// Mitsubishi GX Works2 project: PLC_V3   PLC: FX3G

TYPE ST_STEP : STRUCT
  iEnable : INT;  (* Шаг включён (1 - активен) *)
  iRiseTime : INT;  (* Время подъёма, мин *)
  iHoldTime : INT;  (* Время выдержки, мин *)
  iHoldTempr : INT;  (* Уставка температуры выдержки *)
  iHoldHumid : INT;  (* Уставка влажности выдержки *)
  iVFDSpeed : INT;  (* Скорость ПЧ, % *)
END_STRUCT END_TYPE

TYPE ST_STEPHelper : STRUCT
  iState : INT;  (* Состояние шага: 0 - ожидание, 1 - подъём, 2 - выдержка, 3 - завершено *)
END_STRUCT END_TYPE

TYPE ST_VFD : STRUCT
  xEnable : BOOL;  (* Активация ПЧ (разрешение работы) *)
  xManStart : BOOL;  (* Пуск в ручном режиме *)
  iManSpeed : INT;  (* Скорость в ручном режиме (0-500 = 0.0-50.0 Гц) *)
  iState : INT;  (* Текущее состояние ПЧ (0-3) *)
END_STRUCT END_TYPE

// global labels: GVL
VAR_GLOBAL
  grSteps : ARRAY [0..4] OF ST_STEP;  (* Массив шагов программы сушки (5 шагов) / Назначить R1 как главный *)
  griTLimit AT R31 : INT;  (* Дельта ограничения для ПИД температуры *)
  griHLimit AT R32 : INT;  (* Дельта ограничения для ПИД влажности *)
  griMinVentSpeed AT R33 : INT;  (* Минимальная скорость вентилятора влажности, % *)
  griMinVentDelay AT R34 : INT;  (* Мин. задержка перед включением вентилятора после обнуления ПИД, мин *)
  garstStepHelper : ARRAY [0..4] OF ST_STEPHelper;  (* Массив состояния шагов программы (5 шагов) / Назначить D1090 как главный *)
  grVFD : ARRAY [0..14] OF ST_VFD;  (* Массив ПЧ: [0..13] = ПЧ1-14, [14] = ПЧ ВЕНТ / Назначить M420 D1060 как главный *)
  gxReset AT M400 : BOOL;  (* Сброс *)
  gxStart AT M401 : BOOL;  (* Пуск *)
  gxPIDANTemp AT M402 : BOOL;  (* Включить автонастройку ПИД температуры *)
  gxPIDANHum AT M403 : BOOL;  (* Включить автонастройку ПИД влажности *)
  gxPIDANModeTemp AT M404 : BOOL;  (* 0 - предельный цикл, 1 - ступенчатый отклик *)
  gxPIDANModeHum AT M405 : BOOL;  (* 0 - предельный цикл, 1 - ступенчатый отклик *)
  gxDone AT M406 : BOOL;  (* Процесс сушки завершён *)
  gxAlarmReset AT M407 : BOOL;  (* Сброс аварий *)
  gxProgress AT M408 : BOOL;  (* Процесс сушки выполняется *)
  gxPause AT M409 : BOOL;  (* Процесс сушки на паузе (шаг 40) *)
  gxValve1Work AT M410 : BOOL;  (* Клапан 1 в работе (AO_Valve1 > 0) *)
  gxValve2Work AT M411 : BOOL;  (* Клапан 2 в работе (AO_Valve2 > 0) *)
  gxHasAlarm AT M412 : BOOL;  (* Есть любая зарегистрированная авария *)
  gxNextStep AT M413 : BOOL;  (* Кнопка Следующий этап (HMI) *)
  gxManualMode AT M414 : BOOL;  (* Ручной режим (шаг Idle = 2) *)
  gxFansRun AT M415 : BOOL;  (* Процесс: вентиляторы работают (шаги подъём/выдержка) *)
  giCS_Num AT D1000 : INT;  (* Текущий номер этапа *)
  giCS_RaiseETime AT D1001 : INT;  (* Истекшее время подъёма текущего этапа *)
  giCS_HoldETime AT D1002 : INT;  (* Истекшее время выдержки текущего этапа *)
  giCSVFDSpeed AT D1003 : INT;  (* Скорость ПЧ текущего этапа *)
  giCSTemp_SV AT D1004 : INT;  (* Уставка температуры текущего этапа *)
  giCSHum_SV AT D1005 : INT;  (* Уставка влажности текущего этапа *)
  giCSRaiseTime AT D1006 : INT;  (* Общее время подъёма текущего этапа *)
  giCSHoldTime AT D1007 : INT;  (* Общее время выдержки текущего этапа *)
  giProbeType AT D1008 : INT;  (* Тип датчика температуры: 0 - среднее, 1 - датчик 1, 2 - датчик 2 *)
  giPID_T_SV AT D1009 : INT;  (* ПИД температуры: уставка *)
  giPID_T_PV AT D1010 : INT;  (* ПИД температуры: текущее значение *)
  giPID_T_MV AT D1011 : INT;  (* ПИД температуры: выход (задание на клапаны) *)
  giPID_H_SV AT D1012 : INT;  (* ПИД влажности: уставка *)
  giPID_H_PV AT D1013 : INT;  (* ПИД влажности: текущее значение *)
  giPID_H_MV AT D1014 : INT;  (* ПИД влажности: выход (задание на вентилятор) *)
  giStart_T AT D1015 : INT;  (* Начальная температура для подъёма *)
  giStart_H AT D1016 : INT;  (* Начальная влажность для подъёма *)
  giRaiseET AT D1017 : INT;  (* Остаток времени подъёма, % (0-100) *)
  giHoldET AT D1018 : INT;  (* Остаток времени выдержки, % (0-100) *)
  giCS_NumDisplay AT D1019 : INT;  (* Состояние ПЧ: 0-не активирован, 1-не работает, 2-работает, 3-ошибка *)
  giRaiseMinLeft AT D1020 : INT;  (* Остаток времени подъёма текущего этапа, мин *)
  giHoldMinLeft AT D1021 : INT;  (* Остаток времени выдержки текущего этапа, мин *)
  giValve1Pos AT D1022 : INT;  (* Ручное положение клапана 1 (0-100%) *)
  giValve2Pos AT D1023 : INT;  (* Ручное положение клапана 2 (0-100%) *)
  giPID_T_P AT R503 : INT;  (* ПИД температуры: пропорциональный коэффициент *)
  giPID_T_I AT R504 : INT;  (* ПИД температуры: интегральный коэффициент *)
  giPID_T_D AT R506 : INT;  (* ПИД температуры: дифференциальный коэффициент *)
  giPID_H_P AT R603 : INT;  (* ПИД влажности: пропорциональный коэффициент *)
  giPID_H_I AT R604 : INT;  (* ПИД влажности: интегральный коэффициент *)
  giPID_H_D AT R606 : INT;  (* ПИД влажности: дифференциальный коэффициент *)
END_VAR
VAR_GLOBAL CONSTANT
  c_STATE_IDLE : INT;  (* Состояние: ожидание (0) *)
  c_STATE_RAISE : INT := 1;  (* Состояние: подъём (1) *)
  c_STATE_HOLD : INT := 2;  (* Состояние: выдержка (2) *)
  c_STATE_DONE : INT := 3;  (* Состояние: завершено (3) *)
  c_STEP_NUM : INT := 4;  (* Верхняя граница шагов (4 = 5 шагов 0..4) *)
  c_VFD_ST_NOT_ACTIVE : INT;  (* Состояние ПЧ: не активирован (0) *)
  c_VFD_ST_STOPPED : INT := 1;  (* Состояние ПЧ: не работает (1) *)
  c_VFD_ST_RUNNING : INT := 2;  (* Состояние ПЧ: работает (2) *)
  c_VFD_ST_FAULT : INT := 3;  (* Состояние ПЧ: ошибка (3) *)
END_VAR
VAR_GLOBAL
  AM_ALARMS : ARRAY [0..23] OF ST_AM_ALARM;  (* Хранилище аварий (AlarmManager) *)
  AM_EVENTS : ARRAY [0..0] OF ST_AM_EVENT;  (* Хранилище событий (AlarmManager) *)
END_VAR
VAR_GLOBAL CONSTANT
  c_AM_ALARMS_NUM : INT := 23;  (* Верхняя граница массива аварий = 23 (24 слота) *)
  c_AM_EVENTS_NUM : INT;  (* Верхняя граница массива событий = 0 (1 слот) *)
END_VAR

// global labels: IO
VAR_GLOBAL
  AO_Valve1 AT D8052 : INT;  (* Задание положения клапана 1 (нагрев) *)
  AO_Valve2 AT D8053 : INT;  (* Задание положения клапана 2 (нагрев) *)
  AO_VFD1 AT R23500 : INT;  (* Задание скорости ПЧ1 (0-32000) *)
  AO_VFD2 AT R23501 : INT;  (* Задание скорости ПЧ2 (0-32000) *)
  AO_VFD3 AT R23502 : INT;  (* Задание скорости ПЧ3 (0-32000) *)
  AO_VFD4 AT R23503 : INT;  (* Задание скорости ПЧ4 (0-32000) *)
  AO_VFD5 AT R23504 : INT;  (* Задание скорости ПЧ5 (0-32000) *)
  AO_VFD6 AT R23505 : INT;  (* Задание скорости ПЧ6 (0-32000) *)
  AO_VFD7 AT R23506 : INT;  (* Задание скорости ПЧ7 (0-32000) *)
  AO_VFD8 AT R23507 : INT;  (* Задание скорости ПЧ8 (0-32000) *)
  AO_VFD9 AT R23508 : INT;  (* Задание скорости ПЧ9 (0-32000) *)
  AO_VFD10 AT R23509 : INT;  (* Задание скорости ПЧ10 (0-32000) *)
  AO_VFD11 AT R23510 : INT;  (* Задание скорости ПЧ11 (0-32000) *)
  AO_VFD12 AT R23511 : INT;  (* Задание скорости ПЧ12 (0-32000) *)
  AO_VFD13 AT R23512 : INT;  (* Задание скорости ПЧ13 (0-32000) *)
  AO_VFD14 AT R23513 : INT;  (* Задание скорости ПЧ14 (0-32000) *)
  AO_VFDVent AT R23514 : INT;  (* Задание скорости ПЧ вентиляции/увлажнения (0-32000) *)
  AI_Temp1 AT D0 : INT;  (* Температура 1 в контуре 1 *)
  AI_Temp2 AT D1 : INT;  (* Температура 2 в контуре 1 *)
  AI_Temp3 AT D2 : INT;  (* Температура 1 в контуре 2 *)
  AI_Temp4 AT D3 : INT;  (* Температура 2 в контуре 2 *)
  AI_TempAvg AT D3 : INT;  (* Температура 2 в контуре 2 *)
  AI_TempProd1 AT D4 : INT;  (* Температура продукта 1 *)
  AI_TempProd2 AT D5 : INT;  (* Температура продукта 2 *)
  AI_TempProd3 AT D6 : INT;  (* Температура продукта 3 *)
  AI_TempProdAvg AT D6 : INT;  (* Температура продукта 3 *)
  AI_PVTTempr AT D7 : INT;  (* Температура (ПВТ100) *)
  AI_PVTHumid AT D8 : INT;  (* Влажность (ПВТ100) *)
  AI_Pressure AT D9 : INT;  (* Давление *)
  AI_AirFlow AT D10 : INT;  (* Проток воздуха *)
  AI_Valve1Position AT D11 : INT;  (* Положение клапана 1 (обратная связь) *)
  AI_Valve2Position AT D12 : INT;  (* Положение клапана 2 (обратная связь) *)
  DI_OverheatCP AT X000 : BOOL;  (* Перегрев ЩУ *)
  DI_RKF AT X001 : BOOL;  (* РКФ (ошибка при отсутствии сигнала) *)
  DI_OverheatPU AT X002 : BOOL;  (* Перегрев СШ *)
  DI_VFDAlarm1 AT X003 : BOOL;  (* Ошибка ПЧ1 *)
  DI_VFDAlarm2 AT X004 : BOOL;  (* Ошибка ПЧ2 *)
  DI_VFDAlarm3 AT X005 : BOOL;  (* Ошибка ПЧ3 *)
  DI_VFDAlarm4 AT X006 : BOOL;  (* Ошибка ПЧ4 *)
  DI_VFDAlarm5 AT X007 : BOOL;  (* Ошибка ПЧ5 *)
  DI_VFDAlarm6 AT X010 : BOOL;  (* Ошибка ПЧ6 *)
  DI_VFDAlarm7 AT X011 : BOOL;  (* Ошибка ПЧ7 *)
  DI_VFDAlarm8 AT X012 : BOOL;  (* Ошибка ПЧ8 *)
  DI_VFDAlarm9 AT X020 : BOOL;  (* Ошибка ПЧ9 *)
  DI_VFDAlarm10 AT X021 : BOOL;  (* Ошибка ПЧ10 *)
  DI_VFDAlarm11 AT X022 : BOOL;  (* Ошибка ПЧ11 *)
  DI_VFDAlarm12 AT X023 : BOOL;  (* Ошибка ПЧ12 *)
  DI_VFDAlarm13 AT X024 : BOOL;  (* Ошибка ПЧ13 *)
  DI_VFDAlarm14 AT X025 : BOOL;  (* Ошибка ПЧ14 *)
  DI_VFDAlarmHumid AT X026 : BOOL;  (* Ошибка ПЧ вентиляции/увлажнения *)
  DI_Door AT X030 : BOOL;  (* Дверь открыта *)
  DO_VFD1 AT Y000 : BOOL;  (* Запуск ПЧ1 *)
  DO_VFD2 AT Y001 : BOOL;  (* Запуск ПЧ2 *)
  DO_VFD3 AT Y002 : BOOL;  (* Запуск ПЧ3 *)
  DO_VFD4 AT Y003 : BOOL;  (* Запуск ПЧ4 *)
  DO_VFD5 AT Y004 : BOOL;  (* Запуск ПЧ5 *)
  DO_VFD6 AT Y005 : BOOL;  (* Запуск ПЧ6 *)
  DO_VFD7 AT Y006 : BOOL;  (* Запуск ПЧ7 *)
  DO_VFD8 AT Y007 : BOOL;  (* Запуск ПЧ8 *)
  DO_VFD9 AT Y010 : BOOL;  (* Запуск ПЧ9 *)
  DO_VFD10 AT Y011 : BOOL;  (* Запуск ПЧ10 *)
  DO_VFD11 AT Y012 : BOOL;  (* Запуск ПЧ11 *)
  DO_VFD12 AT Y013 : BOOL;  (* Запуск ПЧ12 *)
  DO_VFD13 AT Y020 : BOOL;  (* Запуск ПЧ13 *)
  DO_VFD14 AT Y021 : BOOL;  (* Запуск ПЧ14 *)
  DO_VFDHum AT Y022 : BOOL;  (* Запуск ПЧ вентиляции/увлажнения *)
  DO_Red AT Y023 : BOOL;  (* Световая колонна: красный *)
  DO_Green AT Y024 : BOOL;  (* Световая колонна: зелёный *)
  DO_Yellow AT Y025 : BOOL;  (* Световая колонна: жёлтый *)
  DO_Buzzer AT Y026 : BOOL;  (* Световая колонна: звук (зуммер) *)
  DO_VFDReset AT Y030 : BOOL;  (* Сброс ошибок ПЧ *)
END_VAR

// task Task_01 (event TRUE, interval 0, priority 31): POU_01
// task INIT (event M8002, interval 0, priority 29): INIT
// task PROCES (event FALSE, interval T#50ms, priority 31): PROCESS
// task TCO (event I650, interval 0, priority 21): 
// user libraries (not included): AlarmManager, Modbus, TimeControl, Utils

PROGRAM POU_01
VAR
  fbAmBlock : FB_AM_IS_BLOCK;  (* Экземпляр FB_AM_IS_BLOCK (проверка блокирующих аварий) *)
  fbTPVentDelay : TP;  (* Таймер задержки выключения вентилятора (TP) *)
  xPIDTEnable : BOOL;  (* Разрешение ПИД температуры *)
  xPIDHEnable : BOOL;  (* Разрешение ПИД влажности *)
  iStep : INT;  (* Текущий шаг/состояние автомата сушки *)
  iCount : INT;  (* Индекс цикла (перебор шагов) *)
  iLastStep : INT;  (* Последний активный шаг *)
END_VAR
fbAmBlock(iProcessNum := 0, iSeverity := 0);

(* Режим работы: ручной = Idle (шаг 2); процесс — рабочие шаги *)
gxManualMode := (iStep = 2);
(* Вентиляторы в процессе работают только на подъёме и выдержке *)
gxFansRun := (iStep = 20 OR iStep = 30);

(* Блокирующая авария — переход в паузу (шаг 40) *)
MOV(fbAmBlock.Q AND iStep > 2, 40, iStep);

(* Кнопка ПУСК отпущена во время подъёма/выдержки — переход в паузу (шаг 40) *)
MOV(NOT gxStart AND (iStep = 20 OR iStep = 30), 40, iStep);

(* Кнопка СБРОС нажата — полный сброс программы (шаг 0), далее Init -> Reset -> Idle *)
MOV(MEP(gxReset), 0, iStep);

(* Кнопка «Следующий этап»: завершить текущий этап и перейти к следующему *)
IF MEP(gxNextStep) AND (iStep = 20 OR iStep = 30) THEN
	garstStepHelper[giCS_Num].iState := c_STATE_DONE;
	giStart_T := grSteps[giCS_Num].iHoldTempr;
	giStart_H := grSteps[giCS_Num].iHoldHumid;
	iStep := 10;
END_IF;

fbTPVentDelay(IN := MEF(DO_VFDHum), PT := F_MIN_TO_TIME(griMinVentDelay));
xPIDTEnable := (iStep = 20 OR iStep = 30) AND (giPID_T_PV < (giPID_T_SV + griTLimit));
xPIDHEnable := (iStep = 20 OR iStep = 30) AND NOT fbTPVentDelay.Q AND (giPID_H_PV > (giPID_H_SV - griHLimit));
PID(xPIDTEnable, giPID_T_SV, giPID_T_PV, R500, giPID_T_MV);
PID(xPIDHEnable, giPID_H_SV, giPID_H_PV, R600, giPID_H_MV);
MOV(NOT xPIDTEnable, 0, giPID_T_MV);
MOV(NOT xPIDHEnable, 0, giPID_H_MV);

CASE iStep OF
	0: (* Init *)
		gxStart := FALSE;
		iStep := 1;

	1: (* Reset *)
		giStart_T := 0;
		giStart_H := 0;
		giCS_Num := 0;
		giCS_RaiseETime := 0;
		giCS_HoldETime := 0;
		giCSVFDSpeed := 0;
		giCSTemp_SV := 0;
		giCSHum_SV := 0;
		giCSRaiseTime := 0;
		giCSHoldTime := 0;
		gxDone := FALSE; gxProgress := FALSE;
		giValve1Pos := 0; giValve2Pos := 0;
		FOR iCount := 0 TO 14 DO
			grVFD[iCount].xManStart := FALSE;
			grVFD[iCount].iManSpeed := 0;
		END_FOR;

		FOR iCount := 0 TO 4 DO
			garstStepHelper[iCount].iState := c_STATE_IDLE;
		END_FOR;
		iStep := 2;

	2: (* Idle *)
		IF gxStart AND NOT fbAmBlock.Q THEN
			(* Сброс ручных команд и уставок при старте процесса *)
			giValve1Pos := 0; giValve2Pos := 0;
			FOR iCount := 0 TO 14 DO
				grVFD[iCount].xManStart := FALSE;
				grVFD[iCount].iManSpeed := 0;
			END_FOR;
			iLastStep := 4;
			FOR iCount := 0 TO 4 DO
				IF grSteps[4 - iCount].iEnable = 1 THEN
					iLastStep := 4 - iCount;
					EXIT;
				END_IF;
			END_FOR;
			IF gxPIDANTemp THEN
				R501 := 2#0000_0000_0011_0001; (* Autotune Step Response *)
				IF NOT gxPIDANModeTemp THEN
					R501 := 2#0000_0000_0111_0001; (* Autotune limit cycle *)
				END_IF;
				gxPIDANTemp := FALSE;
			END_IF;
			IF gxPIDANHum THEN
				R601 := 2#0000_0000_0011_0000; (* Autotune Step Response *)
				IF NOT gxPIDANModeHum THEN
					R601 := 2#0000_0000_0111_0000; (* Autotune limit cycle *)
				END_IF;
				gxPIDANHum := FALSE;
			END_IF;
		
			iStep := 10;
			gxProgress := TRUE;
		END_IF;

	10: (* Step select *)

		FOR iCount := 0 TO 4 DO
			IF grSteps[iCount].iEnable = 1 AND garstStepHelper[iCount].iState < c_STATE_DONE THEN

				(* по умолчанию на подъем начала этапа или востановление подъема,
				но если мы вернулись например после перезагрузки на этап удержания на удержание. *)
				iStep := 20;
				MOV(garstStepHelper[iCount].iState = c_STATE_HOLD, 30, iStep);

				IF iStep > 10 THEN
					giCS_Num := iCount;
					(* Сбрасываем счётчики только если начинаем шаг заново.
					Если возвращаемся в шаг (после паузы/перезагрузки) — сохраняем счёт. *)
					IF garstStepHelper[iCount].iState = c_STATE_IDLE THEN
						giCS_RaiseETime := 0;
						giCS_HoldETime := 0;
					END_IF;
					MOV(iStep = 20, c_STATE_RAISE, garstStepHelper[iCount].iState);
					MOV(iStep = 30, c_STATE_HOLD, garstStepHelper[iCount].iState);
					MOV(giStart_T = 0, giPID_T_PV, giStart_T);
					MOV(giStart_H = 0, giPID_H_PV, giStart_H);
					giCSRaiseTime := grSteps[iCount].iRiseTime;
					giCSHoldTime := grSteps[iCount].iHoldTime;
					giCSTemp_SV := grSteps[iCount].iHoldTempr;
					giCSHum_SV := grSteps[iCount].iHoldHumid;
					giCSVFDSpeed := grSteps[iCount].iVFDSpeed;
					EXIT;
				END_IF;
			END_IF;
		END_FOR;
		MOV(iStep = 10, 50, iStep);


	20: (* Raise *)
		INCP(M8014, giCS_RaiseETime);

		giPID_T_SV := F_SCALE(giCS_RaiseETime, 0, grSteps[giCS_Num].iRiseTime, giStart_T, grSteps[giCS_Num].iHoldTempr);
		giPID_H_SV := F_SCALE(giCS_RaiseETime, 0, grSteps[giCS_Num].iRiseTime, giStart_H, grSteps[giCS_Num].iHoldHumid);

		giRaiseET := F_WORK_LEFT(giCS_RaiseETime, grSteps[giCS_Num].iRiseTime);
		MOV(giCS_RaiseETime >= grSteps[giCS_Num].iRiseTime, 30, iStep);
		MOV(iStep = 30, c_STATE_HOLD, garstStepHelper[giCS_Num].iState);


	30: (* Hold *)
		INCP(M8014, giCS_HoldETime);

		giPID_T_SV := grSteps[giCS_Num].iHoldTempr;
		giPID_H_SV := grSteps[giCS_Num].iHoldHumid;

		giHoldET := F_WORK_LEFT(giCS_HoldETime, grSteps[giCS_Num].iHoldTime);
		MOV(giCS_HoldETime >= grSteps[giCS_Num].iHoldTime, 10, iStep);
		MOV(iStep = 10, c_STATE_DONE, garstStepHelper[giCS_Num].iState);
		MOV(iStep = 10, grSteps[giCS_Num].iHoldTempr, giStart_T);
		MOV(iStep = 10, grSteps[giCS_Num].iHoldHumid, giStart_H);

	40: (* Пауза: выход по повторному включению ПУСК *)
		MOV(gxStart AND NOT fbAmBlock.Q, 10, iStep);

	50: (* Finish *)
		gxDone := TRUE;
		MOV(NOT gxStart, 1, iStep);

END_CASE;

(* Признак паузы для HMI: TRUE, пока автомат находится в шаге 40 *)
gxPause := (iStep = 40);
END_PROGRAM

PROGRAM INIT
VAR
  fbAmInit : FB_AM_INIT;  (* Экземпляр FB_AM_INIT (инициализация аварий) *)
END_VAR
(* Init PID *) (* Настройка параметров ПИД регулирования *)
R500 := 1000; (* Time 1c *)
R501 := 2#0000_0000_0000_0001; (* Heating mode *)
R522 := 4090; (* Output max 100% *)
R523 := 0; (* Output min *)
R525 := 10; (* Delta for Autotune 1.0 C *)
R526 := R522; (* Autotune output upper value *)
R527 := 0; (* Autotune output lower value *)

(* Init PIDHum *) (* Настройка параметров ПИД регулирования *)
R600 := 1000; (* Time 1c *)
R601 := 2#0000_0000_0000_0000; (* Cooling mode *)
R622 := 32000; (* Output max 100% *)
R623 := 0; (* Output min *)
R625 := 10; (* Delta for Autotune 1.0 C *)
R626 := R622; (* Autotune output upper value *)
R627 := 0; (* Autotune output lower value *)

(* Инициализация аварий AlarmManager: 15 ошибок ПЧ (iNum 0..14) *)
fbAmInit(iNum := 0, iSeverity := 0, iProcess := 0, 
    iDelay := 0, xLatch := FALSE, xAutoReset := FALSE, 
    xBuzzer := FALSE, xLock := FALSE);
fbAmInit(iNum := 1);
fbAmInit(iNum := 2);
fbAmInit(iNum := 3);
fbAmInit(iNum := 4);
fbAmInit(iNum := 5);
fbAmInit(iNum := 6);
fbAmInit(iNum := 7);
fbAmInit(iNum := 8);
fbAmInit(iNum := 9);
fbAmInit(iNum := 10);
fbAmInit(iNum := 11);
fbAmInit(iNum := 12);
fbAmInit(iNum := 13);
fbAmInit(iNum := 14);

(* обрывы датчиков *)
fbAmInit(iNum := 15);
fbAmInit(iNum := 16);
fbAmInit(iNum := 17);
fbAmInit(iNum := 18);
fbAmInit(iNum := 19);
fbAmInit(iNum := 20);
fbAmInit(iNum := 21);
fbAmInit(iNum := 22);
fbAmInit(iNum := 23);
END_PROGRAM

PROGRAM PROCESS
VAR
  fbAmSet : FB_AM_SET;  (* Экземпляр FB_AM_SET (регистрация аварий) *)
  fbAmReset : FB_AM_RESET;  (* Экземпляр FB_AM_RESET (сброс аварий) *)
  fbAMPack : FB_AM_PACK_ALARMS;  (* Экземпляр FB_AM_PACK_ALARMS (упаковка аварий в регистры) *)
  fbAmHas : FB_AM_HAS_ALARMS;  (* Экземпляр FB_AM_HAS_ALARMS (наличие любой аварии) *)
  iVFDProcessSpeed : INT;  (* Скорость ПЧ в процессе, 0-32000 (общая для всех ПЧ) *)
END_VAR
CASE giProbeType OF
	0: giPID_T_PV := (AI_Temp1 + AI_Temp2 + AI_Temp3 + AI_Temp4) / 4;
	1: giPID_T_PV := AI_Temp1;
	2: giPID_T_PV := AI_Temp2;
	3: giPID_T_PV := AI_Temp3;
	4: giPID_T_PV := AI_Temp4;
END_CASE;

AI_Temp1 := R23700;
AI_Temp2 := R23701;
AI_Temp3 := R23702;
AI_Temp4 := R23703;
AI_TempAvg := (AI_Temp1 + AI_Temp2 + AI_Temp3 + AI_Temp4) / 4;
AI_TempProd1 := R23704;
AI_TempProd2 := R23705;
AI_TempProd3 := R23706;
AI_TempProdAvg := (AI_TempProd1 + AI_TempProd2 + AI_TempProd3) / 3;
AI_PVTTempr := F_SCALE(R23710, 0, 32000, -400, 800);
AI_PVTHumid := F_SCALE(R23709, 0, 32000, 50, 950);
AI_Pressure := F_SCALE(R23708, 0, 32000, 0, -1000);
AI_AirFlow := F_SCALE(R23711, 0, 32000, 0, 1000);

AI_Valve1Position := F_SCALE(D8032, 0, 4090, 0, 100);
AI_Valve2Position := F_SCALE(D8033, 0, 4090, 0, 100);

giPID_H_PV := AI_PVTHumid;

(* Ручной режим: положение клапанов задаётся с панели (0-100%) *)
AO_Valve1 := SEL(gxManualMode, giPID_T_MV, F_SCALE(giValve1Pos, 0, 100, 0, 4090));
AO_Valve2 := SEL(gxManualMode, giPID_T_MV, F_SCALE(giValve2Pos, 0, 100, 0, 4090));

(* Отображение состояния и положения клапанов (задвижек) на HMI *)
gxValve1Work := AO_Valve1 > 0;
gxValve2Work := AO_Valve2 > 0;


fbAmSet(iNum := 0, xState := DI_VFDAlarm1);
fbAmSet(iNum := 1, xState := DI_VFDAlarm2);
fbAmSet(iNum := 2, xState := DI_VFDAlarm3);
fbAmSet(iNum := 3, xState := DI_VFDAlarm4);
fbAmSet(iNum := 4, xState := DI_VFDAlarm5);
fbAmSet(iNum := 5, xState := DI_VFDAlarm6);
fbAmSet(iNum := 6, xState := DI_VFDAlarm7);
fbAmSet(iNum := 7, xState := DI_VFDAlarm8);
fbAmSet(iNum := 8, xState := DI_VFDAlarm9);
fbAmSet(iNum := 9, xState := DI_VFDAlarm10);
fbAmSet(iNum := 10, xState := DI_VFDAlarm11);
fbAmSet(iNum := 11, xState := DI_VFDAlarm12);
fbAmSet(iNum := 12, xState := DI_VFDAlarm13);
fbAmSet(iNum := 13, xState := DI_VFDAlarm14);
fbAmSet(iNum := 14, xState := DI_VFDAlarmHumid);

(* Обрыв датчиков температуры *)
fbAmSet(iNum := 15, xState := R23700 = -1900); (* Воздух 1 *)
fbAmSet(iNum := 16, xState := R23701 = -1900); (* Воздух 2 *)
fbAmSet(iNum := 17, xState := R23702 = -1900); (* Воздух 3 *)
fbAmSet(iNum := 18, xState := R23703 = -1900); (* Воздух 4 *)
fbAmSet(iNum := 19, xState := R23704 = -1900); (* Продукт 1 *)
fbAmSet(iNum := 20, xState := R23705 = -1900); (* Продукт 2 *)
fbAmSet(iNum := 21, xState := R23706 = -1900); (* Продукт 3 *)
fbAmSet(iNum := 22, xState := D8032 = 32760); (* Положение задвижки ПАР 1 *)
fbAmSet(iNum := 23, xState := D8033 = 32760); (* Положение задвижки ПАР 2 *)

fbAmReset(IN := gxAlarmReset, AutoReset := 60);
fbAMPack(DNUM := 3000, PD := c_AM_PACK_M);

(* Наличие любой аварии (любой процесс/важность) — для HMI *)
fbAmHas(iProcessNum := 0, iSeverity := 0, Q := gxHasAlarm);

DO_VFDReset := gxAlarmReset 
	AND (
		DI_VFDAlarm1
		OR DI_VFDAlarm2
		OR DI_VFDAlarm3
		OR DI_VFDAlarm4
		OR DI_VFDAlarm5
		OR DI_VFDAlarm6
		OR DI_VFDAlarm7
		OR DI_VFDAlarm8
		OR DI_VFDAlarm9
		OR DI_VFDAlarm10
		OR DI_VFDAlarm11
		OR DI_VFDAlarm12
		OR DI_VFDAlarm13
		OR DI_VFDAlarm14
		OR DI_VFDAlarmHumid
	);

iVFDProcessSpeed := F_SCALE(giCSVFDSpeed, 0, 100, 0, 32000);

AO_VFD1 := SEL(gxManualMode, iVFDProcessSpeed, F_SCALE(grVFD[0].iManSpeed, 0, 500, 0, 32000));
DO_VFD1 := grVFD[0].xEnable AND ((gxManualMode AND grVFD[0].xManStart) OR (NOT gxManualMode AND gxFansRun)) AND NOT DI_VFDAlarm1 AND (AO_VFD1 > 0);

AO_VFD2 := SEL(gxManualMode, iVFDProcessSpeed, F_SCALE(grVFD[1].iManSpeed, 0, 500, 0, 32000));
DO_VFD2 := grVFD[1].xEnable AND ((gxManualMode AND grVFD[1].xManStart) OR (NOT gxManualMode AND gxFansRun)) AND NOT DI_VFDAlarm2 AND (AO_VFD2 > 0);

AO_VFD3 := SEL(gxManualMode, iVFDProcessSpeed, F_SCALE(grVFD[2].iManSpeed, 0, 500, 0, 32000));
DO_VFD3 := grVFD[2].xEnable AND ((gxManualMode AND grVFD[2].xManStart) OR (NOT gxManualMode AND gxFansRun)) AND NOT DI_VFDAlarm3 AND (AO_VFD3 > 0);

AO_VFD4 := SEL(gxManualMode, iVFDProcessSpeed, F_SCALE(grVFD[3].iManSpeed, 0, 500, 0, 32000));
DO_VFD4 := grVFD[3].xEnable AND ((gxManualMode AND grVFD[3].xManStart) OR (NOT gxManualMode AND gxFansRun)) AND NOT DI_VFDAlarm4 AND (AO_VFD4 > 0);

AO_VFD5 := SEL(gxManualMode, iVFDProcessSpeed, F_SCALE(grVFD[4].iManSpeed, 0, 500, 0, 32000));
DO_VFD5 := grVFD[4].xEnable AND ((gxManualMode AND grVFD[4].xManStart) OR (NOT gxManualMode AND gxFansRun)) AND NOT DI_VFDAlarm5 AND (AO_VFD5 > 0);

AO_VFD6 := SEL(gxManualMode, iVFDProcessSpeed, F_SCALE(grVFD[5].iManSpeed, 0, 500, 0, 32000));
DO_VFD6 := grVFD[5].xEnable AND ((gxManualMode AND grVFD[5].xManStart) OR (NOT gxManualMode AND gxFansRun)) AND NOT DI_VFDAlarm6 AND (AO_VFD6 > 0);

AO_VFD7 := SEL(gxManualMode, iVFDProcessSpeed, F_SCALE(grVFD[6].iManSpeed, 0, 500, 0, 32000));
DO_VFD7 := grVFD[6].xEnable AND ((gxManualMode AND grVFD[6].xManStart) OR (NOT gxManualMode AND gxFansRun)) AND NOT DI_VFDAlarm7 AND (AO_VFD7 > 0);

AO_VFD8 := SEL(gxManualMode, iVFDProcessSpeed, F_SCALE(grVFD[7].iManSpeed, 0, 500, 0, 32000));
DO_VFD8 := grVFD[7].xEnable AND ((gxManualMode AND grVFD[7].xManStart) OR (NOT gxManualMode AND gxFansRun)) AND NOT DI_VFDAlarm8 AND (AO_VFD8 > 0);

AO_VFD9 := SEL(gxManualMode, iVFDProcessSpeed, F_SCALE(grVFD[8].iManSpeed, 0, 500, 0, 32000));
DO_VFD9 := grVFD[8].xEnable AND ((gxManualMode AND grVFD[8].xManStart) OR (NOT gxManualMode AND gxFansRun)) AND NOT DI_VFDAlarm9 AND (AO_VFD9 > 0);

AO_VFD10 := SEL(gxManualMode, iVFDProcessSpeed, F_SCALE(grVFD[9].iManSpeed, 0, 500, 0, 32000));
DO_VFD10 := grVFD[9].xEnable AND ((gxManualMode AND grVFD[9].xManStart) OR (NOT gxManualMode AND gxFansRun)) AND NOT DI_VFDAlarm10 AND (AO_VFD10 > 0);

AO_VFD11 := SEL(gxManualMode, iVFDProcessSpeed, F_SCALE(grVFD[10].iManSpeed, 0, 500, 0, 32000));
DO_VFD11 := grVFD[10].xEnable AND ((gxManualMode AND grVFD[10].xManStart) OR (NOT gxManualMode AND gxFansRun)) AND NOT DI_VFDAlarm11 AND (AO_VFD11 > 0);

AO_VFD12 := SEL(gxManualMode, iVFDProcessSpeed, F_SCALE(grVFD[11].iManSpeed, 0, 500, 0, 32000));
DO_VFD12 := grVFD[11].xEnable AND ((gxManualMode AND grVFD[11].xManStart) OR (NOT gxManualMode AND gxFansRun)) AND NOT DI_VFDAlarm12 AND (AO_VFD12 > 0);

AO_VFD13 := SEL(gxManualMode, iVFDProcessSpeed, F_SCALE(grVFD[12].iManSpeed, 0, 500, 0, 32000));
DO_VFD13 := grVFD[12].xEnable AND ((gxManualMode AND grVFD[12].xManStart) OR (NOT gxManualMode AND gxFansRun)) AND NOT DI_VFDAlarm13 AND (AO_VFD13 > 0);

AO_VFD14 := SEL(gxManualMode, iVFDProcessSpeed, F_SCALE(grVFD[13].iManSpeed, 0, 500, 0, 32000));
DO_VFD14 := grVFD[13].xEnable AND ((gxManualMode AND grVFD[13].xManStart) OR (NOT gxManualMode AND gxFansRun)) AND NOT DI_VFDAlarm14 AND (AO_VFD14 > 0);


IF gxManualMode THEN
	AO_VFDVent := F_SCALE(grVFD[14].iManSpeed, 0, 500, 0, 32000);
ELSE
	AO_VFDVent := giPID_H_MV;
	(* Если нужно ограничивать, и есть значение приводим его к минимальному. *)
	LIMITATION_E(griMinVentSpeed > 0 AND giPID_H_MV > 0, F_SCALE(griMinVentSpeed, 0, 100, 0, 32000), giPID_H_MV, 32000, AO_VFDVent);
END_IF;
DO_VFDHum := ((gxManualMode AND grVFD[14].xManStart) OR (NOT gxManualMode)) AND NOT DI_VFDAlarmHumid AND (AO_VFDVent > 0);


giCS_NumDisplay := SEL(gxProgress, 0, giCS_Num + 1);

(* Остаток времени текущего этапа в минутах (для HMI) *)
giRaiseMinLeft := LIMITATION(0, giCSRaiseTime - giCS_RaiseETime, giCSRaiseTime);
giHoldMinLeft := LIMITATION(0, giCSHoldTime - giCS_HoldETime, giCSHoldTime);

(* Состояния ПЧ: 0-не активирован, 1-не работает, 2-работает, 3-ошибка *)

IF DI_VFDAlarm1 THEN
	grVFD[0].iState := c_VFD_ST_FAULT;
ELSIF DO_VFD1 THEN
	grVFD[0].iState := c_VFD_ST_RUNNING;
ELSIF grVFD[0].xEnable THEN
	grVFD[0].iState := c_VFD_ST_STOPPED;
ELSE
	grVFD[0].iState := c_VFD_ST_NOT_ACTIVE;
END_IF;

IF DI_VFDAlarm2 THEN
	grVFD[1].iState := c_VFD_ST_FAULT;
ELSIF DO_VFD2 THEN
	grVFD[1].iState := c_VFD_ST_RUNNING;
ELSIF grVFD[1].xEnable THEN
	grVFD[1].iState := c_VFD_ST_STOPPED;
ELSE
	grVFD[1].iState := c_VFD_ST_NOT_ACTIVE;
END_IF;

IF DI_VFDAlarm3 THEN
	grVFD[2].iState := c_VFD_ST_FAULT;
ELSIF DO_VFD3 THEN
	grVFD[2].iState := c_VFD_ST_RUNNING;
ELSIF grVFD[2].xEnable THEN
	grVFD[2].iState := c_VFD_ST_STOPPED;
ELSE
	grVFD[2].iState := c_VFD_ST_NOT_ACTIVE;
END_IF;

IF DI_VFDAlarm4 THEN
	grVFD[3].iState := c_VFD_ST_FAULT;
ELSIF DO_VFD4 THEN
	grVFD[3].iState := c_VFD_ST_RUNNING;
ELSIF grVFD[3].xEnable THEN
	grVFD[3].iState := c_VFD_ST_STOPPED;
ELSE
	grVFD[3].iState := c_VFD_ST_NOT_ACTIVE;
END_IF;

IF DI_VFDAlarm5 THEN
	grVFD[4].iState := c_VFD_ST_FAULT;
ELSIF DO_VFD5 THEN
	grVFD[4].iState := c_VFD_ST_RUNNING;
ELSIF grVFD[4].xEnable THEN
	grVFD[4].iState := c_VFD_ST_STOPPED;
ELSE
	grVFD[4].iState := c_VFD_ST_NOT_ACTIVE;
END_IF;

IF DI_VFDAlarm6 THEN
	grVFD[5].iState := c_VFD_ST_FAULT;
ELSIF DO_VFD6 THEN
	grVFD[5].iState := c_VFD_ST_RUNNING;
ELSIF grVFD[5].xEnable THEN
	grVFD[5].iState := c_VFD_ST_STOPPED;
ELSE
	grVFD[5].iState := c_VFD_ST_NOT_ACTIVE;
END_IF;

IF DI_VFDAlarm7 THEN
	grVFD[6].iState := c_VFD_ST_FAULT;
ELSIF DO_VFD7 THEN
	grVFD[6].iState := c_VFD_ST_RUNNING;
ELSIF grVFD[6].xEnable THEN
	grVFD[6].iState := c_VFD_ST_STOPPED;
ELSE
	grVFD[6].iState := c_VFD_ST_NOT_ACTIVE;
END_IF;

IF DI_VFDAlarm8 THEN
	grVFD[7].iState := c_VFD_ST_FAULT;
ELSIF DO_VFD8 THEN
	grVFD[7].iState := c_VFD_ST_RUNNING;
ELSIF grVFD[7].xEnable THEN
	grVFD[7].iState := c_VFD_ST_STOPPED;
ELSE
	grVFD[7].iState := c_VFD_ST_NOT_ACTIVE;
END_IF;

IF DI_VFDAlarm9 THEN
	grVFD[8].iState := c_VFD_ST_FAULT;
ELSIF DO_VFD9 THEN
	grVFD[8].iState := c_VFD_ST_RUNNING;
ELSIF grVFD[8].xEnable THEN
	grVFD[8].iState := c_VFD_ST_STOPPED;
ELSE
	grVFD[8].iState := c_VFD_ST_NOT_ACTIVE;
END_IF;

IF DI_VFDAlarm10 THEN
	grVFD[9].iState := c_VFD_ST_FAULT;
ELSIF DO_VFD10 THEN
	grVFD[9].iState := c_VFD_ST_RUNNING;
ELSIF grVFD[9].xEnable THEN
	grVFD[9].iState := c_VFD_ST_STOPPED;
ELSE
	grVFD[9].iState := c_VFD_ST_NOT_ACTIVE;
END_IF;

IF DI_VFDAlarm11 THEN
	grVFD[10].iState := c_VFD_ST_FAULT;
ELSIF DO_VFD11 THEN
	grVFD[10].iState := c_VFD_ST_RUNNING;
ELSIF grVFD[10].xEnable THEN
	grVFD[10].iState := c_VFD_ST_STOPPED;
ELSE
	grVFD[10].iState := c_VFD_ST_NOT_ACTIVE;
END_IF;

IF DI_VFDAlarm12 THEN
	grVFD[11].iState := c_VFD_ST_FAULT;
ELSIF DO_VFD12 THEN
	grVFD[11].iState := c_VFD_ST_RUNNING;
ELSIF grVFD[11].xEnable THEN
	grVFD[11].iState := c_VFD_ST_STOPPED;
ELSE
	grVFD[11].iState := c_VFD_ST_NOT_ACTIVE;
END_IF;

IF DI_VFDAlarm13 THEN
	grVFD[12].iState := c_VFD_ST_FAULT;
ELSIF DO_VFD13 THEN
	grVFD[12].iState := c_VFD_ST_RUNNING;
ELSIF grVFD[12].xEnable THEN
	grVFD[12].iState := c_VFD_ST_STOPPED;
ELSE
	grVFD[12].iState := c_VFD_ST_NOT_ACTIVE;
END_IF;

IF DI_VFDAlarm14 THEN
	grVFD[13].iState := c_VFD_ST_FAULT;
ELSIF DO_VFD14 THEN
	grVFD[13].iState := c_VFD_ST_RUNNING;
ELSIF grVFD[13].xEnable THEN
	grVFD[13].iState := c_VFD_ST_STOPPED;
ELSE
	grVFD[13].iState := c_VFD_ST_NOT_ACTIVE;
END_IF;

(* ПЧ вентиляции/увлажнения *)
IF DI_VFDAlarmHumid THEN
	grVFD[14].iState := c_VFD_ST_FAULT;
ELSIF DO_VFDHum THEN
	grVFD[14].iState := c_VFD_ST_RUNNING;
ELSIF grVFD[14].xEnable THEN
	grVFD[14].iState := c_VFD_ST_STOPPED;
ELSE
	grVFD[14].iState := c_VFD_ST_NOT_ACTIVE;
END_IF;
END_PROGRAM
